FUNCTION_BLOCK XeryonDrive
VAR_INPUT
END_VAR
VAR_OUTPUT
	ActPosition : DINT;
	Done : BOOL;
	Busy : BOOL;
	HasError : BOOL;
	HasIndex : BOOL;
	Error : XeryonDriveError;
	MotorOn : BOOL;
	LeftEndstop : BOOL;
	RightEndstop : BOOL;
END_VAR
VAR
	iDriveActualPosition AT %I* : DINT;
	iDriveAmplifiersEnabled AT %I* : BOOL;
	iDriveEndStop AT %I* : BOOL;
	iDriveThermalProtection1 AT %I* : BOOL;
	iDriveThermalProtection2 AT %I* : BOOL;
	iDriveForceZero AT %I* : BOOL;
	iDriveMotorOn AT %I* : BOOL;
	iDriveClosedLoop AT %I* : BOOL;
	iDriveEncoderIndex AT %I* : BOOL;
	iDriveEncoderValid AT %I* : BOOL;
	iDriveSearchingIndex AT %I* : BOOL;
	iDrivePositionReached AT %I* : BOOL;
	iDriveErrorCompensation AT %I* : BOOL;
	iDriveEncoderError AT %I* : BOOL;
	iDriveScanning AT %I* : BOOL;
	iDriveLeftEndStop AT %I* : BOOL;
	iDriveRightEndStop AT %I* : BOOL;
	iDriveErrorLimit AT %I* : BOOL;
	iDriveSearchingOptimalFrequency AT %I* : BOOL;
	iDriveSafetyTimeoutTriggered AT %I* : BOOL;
	iDriveBusy AT %I* : BOOL;
	iDriveEmergencyStop AT %I* : BOOL;
	iDrivePositionFail AT %I* : BOOL;
	iDriveSlot AT %I* : USINT;
	
	qDriveTargetPos AT %Q* : DINT;
	qDriveSpeed AT %Q* : DINT;
	qDriveAcc AT %Q* : INT;
	qDriveDec AT %Q* : INT;
	qCommand AT %Q* : STRING(4);
	qExecute AT %Q* : USINT;
	
	
	new_TargetPos : DINT;
	new_Speed : UDINT;
	new_Acc : INT;
	new_Dec : INT;
	new_command : STRING(4);
	
	state : INT := 0;
	command_start : BOOL;
	command_done : BOOL;
	command_irq : BOOL;
	init_state : INT := -1;
	
	has_index : BOOL;
	
END_VAR

has_index := iDriveEncoderValid;
ActPosition := iDriveActualPosition;
MotorOn := iDriveMotorOn;
LeftEndstop := iDriveLeftEndStop;
RightEndstop := iDriveRightEndStop;
HasIndex := has_index;

// Check error bits
IF(iDriveThermalProtection1) THEN
	HasError := TRUE;
	Error := XeryonDriveError.THERMAL_1;
END_IF
IF(iDriveThermalProtection1) THEN
	HasError := TRUE;
	Error := XeryonDriveError.THERMAL_2;
END_IF
IF(iDriveEncoderError) THEN
	HasError := TRUE;
	Error := XeryonDriveError.ENCODER_ERROR;
END_IF
IF(iDriveEmergencyStop) THEN
	HasError := TRUE;
	Error := XeryonDriveError.ESTOP;
END_IF
IF(iDriveErrorLimit) THEN
	HasError := TRUE;
	Error := XeryonDriveError.ERROR_LIMIT;
END_IF

CASE state OF
	0: // Idle
	 	IF(command_irq = TRUE) THEN
			state := 4;
		END_IF
	 	IF(command_start = TRUE) THEN
			state := 1;
		END_IF
		Busy := FALSE;
	1:
		Busy := TRUE;
		Done := FALSE;
		qCommand := new_command;
		qDriveTargetPos := new_TargetPos;
		qDriveSpeed := UDINT_TO_DINT(new_Speed);
		qDriveAcc := new_Acc;
		qDriveDec := new_Dec;
		qExecute := 255;
		command_start := FALSE;
		command_done := FALSE;
		IF(iDriveBusy = TRUE) THEN
			qExecute := 0;
			state := 2;	
		END_IF		
	2:	
		IF(iDriveBusy = FALSE) THEN
			state := 3;	
		END_IF	
	3: 	IF(command_done = TRUE) THEN
			state := 0;			
			Done := TRUE;
		END_IF
	 	IF(command_irq = TRUE) THEN
			state := 4;
		END_IF
	// Interrupt commands 
	4:	
		command_irq := FALSE;
		Busy := TRUE;
		Done := FALSE;
		qCommand := new_command;
		qDriveTargetPos := new_TargetPos;
		qDriveSpeed := UDINT_TO_DINT(new_Speed);
		qDriveAcc := new_Acc;
		qDriveDec := new_Dec;
		qExecute := 255;
		command_start := FALSE;
		command_done := FALSE;
		IF(iDriveBusy = TRUE) THEN
			qExecute := 0;
			state := 5;	
		END_IF		
	5:	IF(iDriveBusy = FALSE) THEN
			qExecute := 0;
			state := 6;	
		END_IF	
	6:
		state := 0;			
		Done := TRUE;
	
END_CASE

METHOD CheckError : BOOL
VAR_INPUT
END_VAR
CheckError := FALSE;
// Only check these two  bits when moving
IF(iDrivePositionFail) THEN
	HasError := TRUE;
	Error := XeryonDriveError.POS_FAIL;
END_IF
IF(iDriveSafetyTimeoutTriggered) THEN
	HasError := TRUE;
	Error := XeryonDriveError.SAFETY_TIMEOUT;
END_IF
IF(HasError) THEN
	CheckError := TRUE;	
END_IF
END_METHOD

ACTION ClearError:
HasError := FALSE;
Error := XeryonDriveError.NO_ERROR;

// Reset the index when clearing the error
IF(iDriveEncoderValid) THEN
	has_index := TRUE;
ELSE
	has_index := FALSE;
END_IF
END_ACTION

METHOD Enable : XeryonDriveStatus
VAR_INPUT
	val : BOOL;
END_VAR
Enable := XeryonDriveStatus.Waiting;
IF(state = 0) OR (state = 3) THEN
	new_command := 'ENBL';
	IF(val) THEN
		new_TargetPos := 1;
	ELSE
		new_TargetPos := 0;
	END_IF
	command_start := TRUE;
	command_irq := TRUE;
END_IF
IF(state = 6) THEN
	command_done := TRUE;
	Enable := XeryonDriveStatus.Ready;
	// Clear error
	IF(val) THEN
		ClearError();
	END_IF	
END_IF
END_METHOD

METHOD Halt : XeryonDriveStatus
VAR_INPUT
END_VAR
Halt := XeryonDriveStatus.Waiting;
IF(state = 0) OR (state = 3)THEN
	new_command := 'HALT';
	command_start := TRUE;
	command_irq := TRUE;
END_IF
IF(state = 6) THEN
	command_done := TRUE;
	Halt := XeryonDriveStatus.Ready;
END_IF
END_METHOD

METHOD Index : XeryonDriveStatus
VAR_INPUT
	Direction : BOOL;
	Velocity : UDINT;
	Acceleration: UINT;
	Deceleration: UINT;
END_VAR
Index := XeryonDriveStatus.Waiting;
IF(state = 0) THEN
	// Only execute when we don't have an active error
	IF(NOT HasError) THEN
		IF(iDriveAmplifiersEnabled) THEN
			new_command := 'INDX';
			IF(Direction) THEN
				new_TargetPos := +1;	
			ELSE
				new_TargetPos := -1;
			END_IF		
			new_Speed := Velocity;
			new_Acc := UINT_TO_INT(Acceleration);
			new_Dec := UINT_TO_INT(Deceleration);
			command_start := TRUE;
		ELSE
			
			HasError := TRUE;
			IF(NOT iDriveAmplifiersEnabled) THEN
				Error := XeryonDriveError.DRIVE_DISABLED;	
			END_IF		
			Index := XeryonDriveStatus.Error;	
		END_IF
	ELSE
		Index := XeryonDriveStatus.Error;
	END_IF
END_IF
IF(state = 3) THEN
	// Normal flow, when index is found --> ready 
	IF(iDriveEncoderValid) THEN
		command_done := TRUE;
		Index := XeryonDriveStatus.Ready;
	END_IF
	
	// When hitting the endstop signal a SoftError, doesn't need a reset, but limit the motion
	IF(iDriveEndstop) THEN
		command_done := TRUE;
		Index := XeryonDriveStatus.SoftError;		
	END_IF
	
	// Handle drive errors
	IF(CheckError()) THEN
		command_done := TRUE;
		Index := XeryonDriveStatus.Error;
	END_IF
END_IF
IF(state = 6) THEN
	Index := XeryonDriveStatus.Ready;
END_IF
END_METHOD

METHOD Init : BOOL
VAR_IN_OUT
	settings : ARRAY[*] OF XeryonDriveSetting;
END_VAR
Init := FALSE;

// Start
IF(init_state = -1) THEN
	init_state := DINT_TO_INT(LOWER_BOUND(settings, 1));
END_IF

IF(init_state >=  LOWER_BOUND(settings, 1)) AND (init_state < UPPER_BOUND(settings, 1))  THEN
	IF(Write(settings[init_state].setting, settings[init_state].value) <> XeryonDriveStatus.Waiting) THEN
		init_state := init_state + 1;
		IF(init_state = UPPER_BOUND(settings, 1)) THEN
			init_state := -1;
			Init := TRUE;
		END_IF
	END_IF
END_IF
END_METHOD

METHOD MoveAbsolute : XeryonDriveStatus
VAR_INPUT
	Position : DINT;
	Velocity : UDINT;
	Acceleration: UINT;
	Deceleration: UINT;
	
END_VAR
MoveAbsolute := XeryonDriveStatus.Waiting;
IF(state = 0) THEN
	// Only execute when we don't have an active error
	IF(NOT HasError) THEN		
		// Check if we have an index
		IF(has_index) AND iDriveAmplifiersEnabled THEN
			new_command := 'DPOS';
			new_TargetPos := Position;
			new_Speed := Velocity;
			new_Acc := UINT_TO_INT(Acceleration);
			new_Dec := UINT_TO_INT(Deceleration);
			command_start := TRUE;
		ELSE
			HasError := TRUE;
			IF(NOT has_index) THEN
				Error := XeryonDriveError.NO_INDEX;	
			END_IF
			IF(NOT iDriveAmplifiersEnabled) THEN
				Error := XeryonDriveError.DRIVE_DISABLED;	
			END_IF

			MoveAbsolute := XeryonDriveStatus.Error;
		END_IF
	ELSE
		MoveAbsolute := XeryonDriveStatus.Error;
	END_IF	
	
END_IF
IF(state = 3) THEN
	
	// Normal flow, when position is reached  --> ready 
	IF(iDrivePositionReached) THEN
		command_done := TRUE;
		MoveAbsolute := XeryonDriveStatus.Ready;
	END_IF
	
	// When hitting the endstop signal a SoftError, doesn't need a reset, but limit the motion
	IF(iDriveEndstop) THEN
		command_done := TRUE;
		MoveAbsolute := XeryonDriveStatus.SoftError;		
	END_IF
	
	// Handle drive errors
	IF(CheckError()) THEN
		command_done := TRUE;
		MoveAbsolute := XeryonDriveStatus.Error;
	END_IF
	
END_IF
IF(state = 6) THEN
	MoveAbsolute := XeryonDriveStatus.Ready;
END_IF
END_METHOD

METHOD MoveOpen : XeryonDriveStatus
VAR_INPUT
	Direction: BOOL;	
END_VAR
MoveOpen := XeryonDriveStatus.Waiting;
IF(state = 0) THEN
	IF( NOT HasError) THEN
		IF iDriveAmplifiersEnabled THEN
			new_command := 'MOVE';
			IF(Direction) THEN
				new_TargetPos := +1;	
			ELSE
				new_TargetPos := -1;
			END_IF
			new_Speed := 0;
			new_Acc := UINT_TO_INT(0);
			new_Dec := UINT_TO_INT(0);
			command_start := TRUE;
		ELSE
			HasError := TRUE;
			IF(NOT iDriveAmplifiersEnabled) THEN
				Error := XeryonDriveError.DRIVE_DISABLED;	
			END_IF		
			MoveOpen := XeryonDriveStatus.Error;	
		END_IF
	ELSE
		MoveOpen := XeryonDriveStatus.Error;
	END_IF	
END_IF
IF(state = 3) THEN
	command_done := TRUE;
	MoveOpen := XeryonDriveStatus.Ready;
END_IF
IF(state = 6) THEN
	MoveOpen := XeryonDriveStatus.Ready;
END_IF
END_METHOD

METHOD Reset : XeryonDriveStatus
VAR_INPUT
END_VAR
Reset := XeryonDriveStatus.Waiting;
IF(state = 0) OR (state = 3) THEN
	new_command := 'RSET';
	command_start := TRUE;
	command_irq := TRUE;
END_IF
IF(state = 6) THEN
	command_done := TRUE;
	Reset := XeryonDriveStatus.Ready;
	
	// Clear errors
	ClearError();
	
	// Clear Index
	has_index := FALSE;
	
END_IF
END_METHOD

METHOD ResetEncoder : XeryonDriveStatus
ResetEncoder := XeryonDriveStatus.Waiting;
IF(state = 0) OR (state = 3) THEN
	new_command := 'ENCR';
	command_start := TRUE;
	command_irq := TRUE;
END_IF
IF(state = 6) THEN
	command_done := TRUE;
	ResetEncoder := XeryonDriveStatus.Ready;
	
	// Clear Index
	has_index := FALSE;
	
END_IF
END_METHOD

METHOD Scan : XeryonDriveStatus
VAR_INPUT
	Direction: BOOL;
	Velocity : UDINT;
	Acceleration: UINT;
	Deceleration: UINT;
END_VAR
Scan := XeryonDriveStatus.Waiting;
IF(state = 0) THEN
	IF( NOT HasError) THEN
		IF iDriveAmplifiersEnabled THEN
			new_command := 'SCAN';
			IF(Direction) THEN
				new_TargetPos := +1;	
			ELSE
				new_TargetPos := -1;
			END_IF
			new_Speed := Velocity;
			new_Acc := UINT_TO_INT(Acceleration);
			new_Dec := UINT_TO_INT(Deceleration);
			command_start := TRUE;
		ELSE
			HasError := TRUE;
			IF(NOT iDriveAmplifiersEnabled) THEN
				Error := XeryonDriveError.DRIVE_DISABLED;	
			END_IF		
			Scan := XeryonDriveStatus.Error;	
		END_IF
	ELSE
		Scan := XeryonDriveStatus.Error;
	END_IF	
END_IF
IF(state = 3) THEN
	// Normal flow, when end stop is reached  --> ready 
	IF(((new_TargetPos = +1) AND (iDriveRightEndStop)) OR 
	   ((new_TargetPos = -1) AND (iDriveLeftEndStop))) THEN
		command_done := TRUE;
		Scan := XeryonDriveStatus.Ready;
	END_IF
	
	// Handle drive errors
	IF(CheckError()) THEN
		command_done := TRUE;
		Scan := XeryonDriveStatus.Error;
	END_IF	
END_IF
IF(state = 6) THEN
	Scan := XeryonDriveStatus.Ready;
END_IF
END_METHOD

METHOD Stop : XeryonDriveStatus
VAR_INPUT
END_VAR
Stop := XeryonDriveStatus.Waiting;
IF(state = 0) OR (state = 3) THEN
	new_command := 'STOP';
	command_start := TRUE;
	command_irq := TRUE;
END_IF
IF(state = 6) THEN
	command_done := TRUE;
	Stop := XeryonDriveStatus.Ready;
	
END_IF
END_METHOD

METHOD Write : XeryonDriveStatus
VAR_INPUT
	setting : STRING(4);
	value : DINT;
END_VAR
Write := XeryonDriveStatus.Waiting;
IF(state = 0) THEN
	new_command := setting;
	new_TargetPos := value;
	new_Speed := 0;
	new_Acc := 0;
	new_Dec := 0;
	command_start := TRUE;
END_IF
IF(state = 3) THEN
	command_done := TRUE;
	Write := XeryonDriveStatus.Ready;
END_IF
END_METHOD

END_FUNCTION_BLOCK

(* stored: Version 1.1.0.1, ProductVersion 3.1.4024.16
   POU XeryonDrive: Id {6903b1ac-34a8-4f18-b448-c4393b0e95e9}, SpecialFunc None
   Method CheckError: Id {be3ec597-8321-4986-b5a2-d4320c676b8c}
   Action ClearError: Id {33d562a0-ef5b-4301-911a-9442b0c91ea4}
   Method Enable: Id {a3b6ceb4-20a9-48fa-ae69-fc1fa186446f}
   Method Halt: Id {9d6801bf-8859-498b-bd0a-a0b58bb4cdd3}
   Method Index: Id {d7a89949-eead-4162-9511-56dbdd6b904a}
   Method Init: Id {f8435b93-3b45-4ef3-aaf8-528b808b54c0}
   Method MoveAbsolute: Id {cac29e84-f0d7-404f-8481-4bac1dfb823e}
   Method MoveOpen: Id {5bec61eb-be64-4112-abbf-9f8c73e6c1d7}
   Method Reset: Id {9ecb55c1-cf98-4bc6-aa47-2e4653aaefc2}
   Method ResetEncoder: Id {69a5e7ad-7b3e-45ee-9780-0a83108bbff8}
   Method Scan: Id {d3f14fe7-6bfa-4065-895d-33345dc131cf}
   Method Stop: Id {5ef57abf-1ef2-43a2-b21e-791191a45540}
   Method Write: Id {3e18ae05-e84d-4962-b1be-392337d645bc} *)
